INTERFACE ITF_BaseGroupElement_HMI_Connector EXTENDS 
		ITF_BaseGroupElement_HMI_Connector_View, ITF_BaseGroupElement_HMI_Connector_Command

END_INTERFACE

(* stored: Version 1.1.0.1
   Itf ITF_BaseGroupElement_HMI_Connector: Id {05989430-ed19-0f83-3f5e-45021d208310} *)
